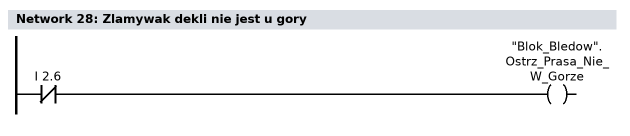
NETWORK
TITLE = Zlamywak dekli nie jest u gory 
      AN    I 2.6;
      =     "Blok_Bledow".Ostrz_Prasa_Nie_W_Gorze;
END_FUNCTION

FUNCTION "FC_HMI" : VOID	// FC 120
VERSION : 0.1
VAR_TEMP
  LW0_Help : INT ;
END_VAR
BEGIN
NETWORK
TITLE =
//Ten network celowo wolny
NETWORK
TITLE = Tryb Pracy Wiazanie poprzeczne
//Wybranie trybu pracy resetuje pozostale tryby pracy
//1-Przelot
      A     "DB_HMI".HMI_IN_OUT.Tp_Przelot;
      R     "DB_HMI".HMI_IN_OUT.Tp_Wiazanie_Poprzeczne;
      R     "DB_HMI".HMI_IN_OUT.Tp_Wiazanie_Wzdluzne;
      R     "DB_HMI".HMI_IN_OUT.Tp_Wiazanie_Pop_Wzdl;
      R     "Blok_Para".Wiazanie_Poprzeczne;
      R     "Blok_Para".Wiazanie_Wzdluzne;
NETWORK
TITLE = Tryb Pracy Wiazanie poprzeczne
//Wybranie trybu pracy resetuje pozostale tryby pracy
//2-Wiazanie Poprzeczne
      A     "DB_HMI".HMI_IN_OUT.Tp_Wiazanie_Poprzeczne;
      R     "DB_HMI".HMI_IN_OUT.Tp_Przelot;
      R     "DB_HMI".HMI_IN_OUT.Tp_Wiazanie_Wzdluzne;
      R     "DB_HMI".HMI_IN_OUT.Tp_Wiazanie_Pop_Wzdl;
      S     "Blok_Para".Wiazanie_Poprzeczne;
      R     "Blok_Para".Wiazanie_Wzdluzne;
NETWORK
TITLE = Tryb Pracy Wiazanie poprzeczne
//Wybranie trybu pracy resetuje pozostale tryby pracy
//3-Wiazanie Wzdluzne
      A     "DB_HMI".HMI_IN_OUT.Tp_Wiazanie_Wzdluzne;
      R     "DB_HMI".HMI_IN_OUT.Tp_Przelot;
      R     "DB_HMI".HMI_IN_OUT.Tp_Wiazanie_Poprzeczne;
      R     "DB_HMI".HMI_IN_OUT.Tp_Wiazanie_Pop_Wzdl;
      R     "Blok_Para".Wiazanie_Poprzeczne;
      S     "Blok_Para".Wiazanie_Wzdluzne;
NETWORK
TITLE = Tryb Pracy Wiazanie poprzeczne
//Wybranie trybu pracy resetuje pozostale tryby pracy
//4-Wiazanie Poprzeczne i wzdluzne
      A     "DB_HMI".HMI_IN_OUT.Tp_Wiazanie_Pop_Wzdl;
      R     "DB_HMI".HMI_IN_OUT.Tp_Przelot;
      R     "DB_HMI".HMI_IN_OUT.Tp_Wiazanie_Poprzeczne;
      R     "DB_HMI".HMI_IN_OUT.Tp_Wiazanie_Wzdluzne;
      S     "Blok_Para".Wiazanie_Poprzeczne;
      S     "Blok_Para".Wiazanie_Wzdluzne;
NETWORK
TITLE = wybrano tryb pracy przelot
      AN    "Blok_Para".Wiazanie_Wzdluzne;
      AN    "Blok_Para".Wiazanie_Poprzeczne;
      =     "DB_HMI".HMI_IN.Wybrano_TP_Przelot;
//-wzdl
      A     "Blok_Para".Wiazanie_Wzdluzne;
      AN    "Blok_Para".Wiazanie_Poprzeczne;
      =     "DB_HMI".HMI_IN.Wybrano_TP_Wiazanie_Wzdl;
//-pop
      AN    "Blok_Para".Wiazanie_Wzdluzne;
      A     "Blok_Para".Wiazanie_Poprzeczne;
      =     "DB_HMI".HMI_IN.Wybrano_TP_Wiazanie_Pop;
//-pop -wzdl
      A     "Blok_Para".Wiazanie_Wzdluzne;
      A     "Blok_Para".Wiazanie_Poprzeczne;
      =     "DB_HMI".HMI_IN.Wybrano_TP_Wiazanie_Krzy;
NETWORK
TITLE =
//znacznik trybu wiazania
//krok_1  - przelot
      A     "DB_HMI".HMI_IN.Wybrano_TP_Przelot;
      L     1;
      JC    ztw;
//krok_2 - wzdluzna
      A     "DB_HMI".HMI_IN.Wybrano_TP_Wiazanie_Wzdl;
      L     2;
      JC    ztw;
//krok_3 - poprzeczne
      A     "DB_HMI".HMI_IN.Wybrano_TP_Wiazanie_Pop;
      L     3;
      JC    ztw;
//krok_4 - krzyzowe
      A     "DB_HMI".HMI_IN.Wybrano_TP_Wiazanie_Krzy;
      L     4;
      JC    ztw;
//daj 0
ztw:  T     "DB_HMI".HMI_IN.tryb_wiaz;
NETWORK
TITLE = Tryb Pracy Wiazanie wzduzne
//Zalaczenie Pozycjonowania
      A     "DB_HMI".HMI_IN_OUT.Tp_Pozycjonowanie;
      S     "Blok_Para".Pozycjonowanie;
      AN    "DB_HMI".HMI_IN_OUT.Tp_Pozycjonowanie;
      R     "Blok_Para".Pozycjonowanie;
      NOP   0;
NETWORK
TITLE = fotokomorka hamowania obrotnicy do kata 0st
//Fotokomorki katow pozycjonowania obrotnicy
      A     "AIO".Czuj_19_B.Czujnik_Ham_0_St;
      =     "DB_HMI".HMI_IN.Czujnik_Ham_0_St;
      A     "AIO".Czuj_19_B.Czujnik_0_St;
      =     "DB_HMI".HMI_IN.Czujnik_0_St;
      A     "AIO".Czuj_19_B.Czujnik_Ham_90_St;
      =     "DB_HMI".HMI_IN.Czujnik_Ham_90_St;
      A     "AIO".Czuj_19_B.Czujnik_90_St;
      =     "DB_HMI".HMI_IN.Czujnik_90_St;
      A     "AIO".Czuj_17_B.Czujnik_Ham_180_St;
      =     "DB_HMI".HMI_IN.Czujnik_Ham_180_St;
      A     "AIO".Czuj_17_B.Czujnik_180_St;
      =     "DB_HMI".HMI_IN.Czujnik_180_St;
      A     "AIO".Czuj_17_B.Czujnik_Ham_270_St;
      =     "DB_HMI".HMI_IN.Czujnik_Ham_270_St;
      A     "AIO".Czuj_17_B.Czujnik_270_St;
      =     "DB_HMI".HMI_IN.Czujnik_270_St;
NETWORK
TITLE = foto przednie bandzie wlotowej
//Fotokommorki
      A     "AIO".Banda_23.Foto_1;
      =     "DB_HMI".HMI_IN.Foto_Tasma_1_Przod;
      A     "AIO".Banda_23.Foto_2;
      =     "DB_HMI".HMI_IN.Foto_Tasma_1_Tyl;
      A     "AIO".Banda_24.Foto_1;
      =     "DB_HMI".HMI_IN.Foto_Tasma_2_Przod;
      A     "AIO".Banda_24.Foto_2;
      =     "DB_HMI".HMI_IN.Foto_Tasma_2_Tyl;
      A     "AIO".Obr_15.Foto_1;
      =     "DB_HMI".HMI_IN.Foto_Obrotnica_3_Przod;
      A     "AIO".Obr_15.Foto_2;
      =     "DB_HMI".HMI_IN.Foto_Obrotnica_3_Tyl;
      A     "AIO".Banda_2.Foto_1;
      =     "DB_HMI".HMI_IN.Foto_Tasma_4_Przod;
      A     "AIO".Banda_2.Foto_2;
      =     "DB_HMI".HMI_IN.Foto_Tasma_4_Tyl;
NETWORK
TITLE = tasma 1
//do wizualizacji przemieszczania palety na tasmie 1
      AN    "AIO".Banda_23.Foto_1;
      A     "AIO".Banda_23.Foto_2;
      =     "DB_HMI".HMI_IN.Paleta_na_Tasmie_1_T;
      A     "AIO".Banda_23.Foto_1;
      AN    "AIO".Banda_23.Foto_2;
      AN    "AIO".Banda_24.Foto_2;
      =     "DB_HMI".HMI_IN.Paleta_na_Tasmie_1_P;
      A     "AIO".Banda_23.Foto_1;
      A     "AIO".Banda_23.Foto_2;
      =     "DB_HMI".HMI_IN.Paleta_na_Tasmie_1;
NETWORK
TITLE = tasma 2
//do wizualizacji przemieszczania palety na tasmie 2
      AN    "AIO".Banda_24.Foto_1;
      A     "AIO".Banda_24.Foto_2;
      =     "DB_HMI".HMI_IN.Paleta_na_Tasmie_2_T;
      A     "AIO".Banda_24.Foto_1;
      AN    "AIO".Banda_24.Foto_2;
      AN    "AIO".Obr_15.Foto_1;
      =     "DB_HMI".HMI_IN.Paleta_na_Tasmie_2_P;
      A     "AIO".Banda_24.Foto_1;
      A     "AIO".Banda_24.Foto_2;
      =     "DB_HMI".HMI_IN.Paleta_na_Tasmie_2;
NETWORK
TITLE = tasma 3 (obrotnica)
//do wizualizacji przemieszczania palety na tasmie 3
      A     "AIO".Obr_15.Foto_1;
      AN    "AIO".Obr_15.Foto_2;
      A     "DB_HMI".HMI_IN.Czujnik_0_St;
      =     "DB_HMI".HMI_IN.Paleta_na_Tasmie_3_T;
      AN    "AIO".Obr_15.Foto_1;
      A     "AIO".Obr_15.Foto_2;
      AN    "AIO".Banda_2.Foto_2;
      A     "DB_HMI".HMI_IN.Czujnik_0_St;
      =     "DB_HMI".HMI_IN.Paleta_na_Tasmie_3_P;
      A     "AIO".Obr_15.Foto_1;
      A     "AIO".Obr_15.Foto_2;
      A(;
      O     "DB_HMI".HMI_IN.Czujnik_0_St;
      O     "DB_HMI".HMI_IN.Czujnik_180_St;
      );
      =     "DB_HMI".HMI_IN.Paleta_na_Tasmie_3_0_180;
      A     "AIO".Obr_15.Foto_1;
      A     "AIO".Obr_15.Foto_2;
      A(;
      O     "DB_HMI".HMI_IN.Czujnik_90_St;
      O     "DB_HMI".HMI_IN.Czujnik_270_St;
      );
      =     "DB_HMI".HMI_IN.Paleta_na_Tasmie_3_90_27;
NETWORK
TITLE = tasma 4
//do wizualizacji przemieszczania palety na tasmie 4
      AN    "AIO".Banda_2.Foto_1;
      A     "AIO".Banda_2.Foto_2;
      =     "DB_HMI".HMI_IN.Paleta_na_Tasmie_4_T;
      A     "AIO".Banda_2.Foto_1;
      AN    "AIO".Banda_2.Foto_2;
      =     "DB_HMI".HMI_IN.Paleta_na_Tasmie_4_P;
      A     "AIO".Banda_2.Foto_1;
      A     "AIO".Banda_2.Foto_2;
      =     "DB_HMI".HMI_IN.Paleta_na_Tasmie_4;
NETWORK
TITLE = motor obrotnica 3 counter clock wise
//Napedy band
      A     "AIO".Obr_15.CC_Wise;
      =     "DB_HMI".HMI_IN.Motor_Obrotnica_3_CCW;
      A     "AIO".Obr_15.C_Wise;
      =     "DB_HMI".HMI_IN.Motor_Obrotnica_3_CW;
      A     "AIO".Banda_23.CC_Wise;
      =     "DB_HMI".HMI_IN.Motor_Tasma_1_Przod;
      A     "AIO".Banda_23.C_Wise;
      =     "DB_HMI".HMI_IN.Motor_Tasma_1_Tyl;
      A     "AIO".Banda_24.C_Wise;
      =     "DB_HMI".HMI_IN.Motor_Tasma_2_Przod;
      A     "AIO".Banda_24.CC_Wise;
      =     "DB_HMI".HMI_IN.Motor_Tasma_2_Tyl;
      A     "AIO".Banda_1.C_Wise;
      =     "DB_HMI".HMI_IN.Motor_Tasma_3_Przod;
      A     "AIO".Banda_1.CC_Wise;
      =     "DB_HMI".HMI_IN.Motor_Tasma_3_Tyl;
      A     "AIO".Banda_2.CC_Wise;
      =     "DB_HMI".HMI_IN.Motor_Tasma_4_Przod;
      A     "AIO".Banda_2.C_Wise;
      =     "DB_HMI".HMI_IN.Motor_Tasma_4_Tyl;
NETWORK
TITLE = obwod bezpieczenstwa bindownicy
//sygnaly wymiany danych pomiedzy transportem palet a bindownica
      A     I 2.0;
      =     "DB_HMI".HMI_IN.Interfefs_B_do_TP_B1;
      A     I 2.1;
      =     "DB_HMI".HMI_IN.Interfefs_B_do_TP_B2;
      A     I 2.3;
      =     "DB_HMI".HMI_IN.Interfefs_B_do_TP_B3;
      A     I 2.4;
      =     "DB_HMI".HMI_IN.Interfefs_B_do_TP_B4;
      A     I 2.2;
      =     "DB_HMI".HMI_IN.Interfefs_B_do_TP_B5;
//Transport do bindownicy 
      A     M 6.3;
      =     "DB_HMI".HMI_IN.Interfefs_TP_do_B_TP1;
      A     Q 1.1;
      =     "DB_HMI".HMI_IN.Interfefs_TP_do_B_TP2;
      A     Q 1.2;
      =     "DB_HMI".HMI_IN.Interfefs_TP_do_B_TP3;
NETWORK
TITLE = przycisk zalaczenie Strefy bezpieczenstwa
//przyciski, przelaczniki kierunkow i lampki na panelu
      A     I 0.0;
      =     "DB_HMI".HMI_IN.PB_Strefa_bezpieczenstwa;
      A     I 0.1;
      =     "DB_HMI".HMI_IN.PB_Reczny;
      A     I 0.2;
      =     "DB_HMI".HMI_IN.PB_Auto;
      A     I 0.3;
      =     "DB_HMI".HMI_IN.PB_Reset;
      A     I 0.4;
      =     "DB_HMI".HMI_IN.PB_Stop;
      A     I 0.5;
      =     "DB_HMI".HMI_IN.PB_Cykl_Start;
      A     I 0.6;
      =     "DB_HMI".HMI_IN.PB_Tasma1_Tyl;
      A     I 0.7;
      =     "DB_HMI".HMI_IN.PB_Tasma1_Przod;
      A     I 1.0;
      =     "DB_HMI".HMI_IN.PB_Tasma2_Tyl;
      A     I 1.1;
      =     "DB_HMI".HMI_IN.PB_Tasma2_Przod;
      A     I 1.2;
      =     "DB_HMI".HMI_IN.PB_Tasma3_Tyl;
      A     I 1.3;
      =     "DB_HMI".HMI_IN.PB_Tasma3_Przod;
      A     I 1.4;
      =     "DB_HMI".HMI_IN.PB_Tasma4_Tyl;
      A     I 1.5;
      =     "DB_HMI".HMI_IN.PB_Tasma4_Przod;
      A     I 1.6;
      =     "DB_HMI".HMI_IN.PB_Tasma3_Obr_CW;
      A     I 1.7;
      =     "DB_HMI".HMI_IN.PB_Tasma3_Obr_CCW;
      A     Q 0.0;
      =     "DB_HMI".HMI_IN.Lampka_Blad_Bind;
      A     Q 0.1;
      =     "DB_HMI".HMI_IN.Lampka_Strzal_Tasmy;
      A     Q 0.2;
      =     "DB_HMI".HMI_IN.Lampka_Strefa_Bezp;
      A     Q 0.3;
      =     "DB_HMI".HMI_IN.Lampka_PB_Reczny;
      A     Q 0.4;
      =     "DB_HMI".HMI_IN.Lampka_PB_Auto;
      A     Q 0.5;
      =     "DB_HMI".HMI_IN.Lampka_PB_Reset;
      A     Q 0.6;
      =     "DB_HMI".HMI_IN.Lampka_PB_Stop;
      A     Q 0.7;
      =     "DB_HMI".HMI_IN.Lampka_PB_Cykl_Start;
NETWORK
TITLE =
//Start/Stop calej lini
      A     "DB_HMI".HMI_OUT.Start_Lini_z_OP;
      =     "Blok_Para".Start_Lini_z_OP;
      A     "DB_HMI".HMI_OUT.Stop_Lini_z_OP;
      =     "Blok_Para".Stop_Lini_z_OP;
NETWORK
TITLE = //wyjazd wtrybie auto
//Wyzwolenie wyjazdu palety gdy paleta stoi na bandzie obrotowej a nie wyjezdza
//
      A     "DB_HMI".HMI_OUT.Wyzwolenie_Wyjazdu;
      =     "Blok_Para".Trigger_Wyjazd;
NETWORK
TITLE = Znacznik stanu kurtyny optycznej na wlocie
//Bariery optyczne bindownicy
      AN    "AIO".Kurtyna_25.OSSD_Tor_1_1;
      AN    "AIO".Kurtyna_25.OSSD_Tor_1_2;
      AN    "AIO".Kurtyna_25.OSSD_Tor_2_1;
      AN    "AIO".Kurtyna_25.OSSD_Tor_2_2;
      =     "DB_HMI".HMI_IN.Kurtyna_Wlot_Ok;
      AN    "AIO".Kurtyna_26.OSSD_Tor_1_1;
      AN    "AIO".Kurtyna_26.OSSD_Tor_1_2;
      AN    "AIO".Kurtyna_26.OSSD_Tor_2_1;
      AN    "AIO".Kurtyna_26.OSSD_Tor_2_2;
      =     "DB_HMI".HMI_IN.Kurtyna_Wylot_Ok;
      A     M 6.2;
      =     "DB_HMI".HMI_IN.Rygiel;
NETWORK
TITLE = Znacznik pracy calej linii transportowej
      A     Q 8.3;
      =     "DB_HMI".HMI_IN.Linia_transportowa_praca;
NETWORK
TITLE = tryb pracy bindownicy: Auto(1) Reczny(0)
      A     "Blok_Bledow_Program".Blad_Krok_1;
      =     "DB_HMI".HMI_IN.Krok_1;
      A     "Blok_Bledow_Program".Blad_Krok_2;
      =     "DB_HMI".HMI_IN.Krok_2;
      A     "Blok_Bledow_Program".Blad_Krok_3;
      =     "DB_HMI".HMI_IN.Krok_3;
      A     "Blok_Bledow_Program".Blad_Krok_4;
      =     "DB_HMI".HMI_IN.Krok_4;
      A     "Blok_Bledow_Program".Blad_Krok_5;
      =     "DB_HMI".HMI_IN.Krok_5;
      A     "Blok_Bledow_Program".Blad_Krok_6;
      =     "DB_HMI".HMI_IN.Krok_6;
NETWORK
TITLE =
//przypisanie stanu wejsc i wyjsc
      L     IB 0;
      T     "DB_HMI".HMI_IN.input_0;
      L     IB 1;
      T     "DB_HMI".HMI_IN.input_1;
      L     IB 2;
      T     "DB_HMI".HMI_IN.input_2;
      L     IB 3;
      T     "DB_HMI".HMI_IN.input_3;
      L     QB 0;
      T     "DB_HMI".HMI_IN.output_0;
      L     QB 1;
      T     "DB_HMI".HMI_IN.output_1;
      L     QB 2;
      T     "DB_HMI".HMI_IN.output_2;
      L     QB 3;
      T     "DB_HMI".HMI_IN.output_3;
      L     IB 8;
      T     "DB_HMI".HMI_IN.input_8;
      L     IB 9;
      T     "DB_HMI".HMI_IN.input_9;
      L     IB 10;
      T     "DB_HMI".HMI_IN.input_10;
      L     IB 11;
      T     "DB_HMI".HMI_IN.input_11;
NETWORK
TITLE = krok 1 trybu pracy
//Przypisanie aktualnych krokow 
//krok_1  - jedz na pozycje 
      A     "Blok_Para".Krok_1;
      L     1;
      JC    tr;
//krok_2 - szukaj srodka 
      A     "Blok_Para".krok_2;
      L     2;
      JC    tr;
//krok_3 - jedz na prawo
      A     "Blok_Para".krok_3;
      L     3;
      JC    tr;
//krok_4 - strzelaj 
      A     "Blok_Para".krok_4;
      L     4;
      JC    tr;
//krok_5  - pauza po strzale
      A     "Blok_Para".krok_5;
      L     5;
      JC    tr;
//krok_6 - jedz do srodka
      A     "Blok_Para".krok_6;
      L     6;
      JC    tr;
//daj 0
      L     0;
tr:   T     "DB_HMI".HMI_IN.INT_Liczba_Akt_Kroku;
NETWORK
TITLE = znacznik migania bledu
//Sprawdzenie czy sa bledy jak sa to miganie bledow
      SET;
      R     "DB_HMI".HMI_IN.Znacznik_Migania_Bledu;
      O(;
      L     DB119.DBD 0;
      L     0;
      <>D;
      );
      O(;
      L     DB119.DBD 4;
      L     0;
      <>D;
      );
      O(;
      L     DB119.DBD 8;
      L     0;
      <>D;
      );
      S     "DB_HMI".HMI_IN.Znacznik_Migania_Bledu;
NETWORK
TITLE = czujnik prasy s 22
//Obsluga wygladu prasy
//
      A     I 2.6;
      =     "DB_HMI".HMI_IN.Czujnik_Prasa;
//zawor prasa
      AN    Q 1.0;
      =     "DB_HMI".HMI_IN.Stan_Zaworu;
NETWORK
TITLE =
//Aktualizacja godziny/daty panela z godzina/czasem PLC
      CALL  "READ_CLK" (
           RET_VAL                  := #LW0_Help,
           CDT                      := "DB_HMI".HMI_IN.Aktualna_Data);
END_FUNCTION

FUNCTION "Funkcja_Zegara" : VOID	// FC 140
AUTHOR : Kng
NAME : HELP_FC
VERSION : 0.1
VAR_INPUT
  Timer_NR : TIMER ;
  Czas : S5TIME ;
END_VAR
VAR_IN_OUT
  Wyjscie : BOOL ;
END_VAR
BEGIN
NETWORK
TITLE =
      A     #Timer_NR;
      SAVE;
      NOT;
      L     #Czas;
      SD    #Timer_NR;
      X     BR;
      X     #Wyjscie;
      =     #Wyjscie;
END_FUNCTION

DATA_BLOCK DB 4
VERSION : 0.0
"Czesc_Bindujaca"
BEGIN
END_DATA_BLOCK

DATA_BLOCK DB 5
VERSION : 0.0
"Czesc_Trasnportujaca"
BEGIN
END_DATA_BLOCK

DATA_BLOCK "AIO"	// DB 10
VERSION : 0.1
  STRUCT
   Banda_1 : UDT 1;	//Temporary placeholder variable
   Banda_2 : UDT 1;
   Banda_3 : UDT 1;
   Banda_4 : UDT 9;
   Banda_5 : UDT 1;
   Banda_6 : UDT 1;
   Banda_7 : UDT 1;
   Banda_8 : UDT 1;
   Banda_9 : UDT 1;
   Banda_10 : UDT 1;
   Banda_11 : UDT 1;
   Banda_12 : UDT 1;
   Banda_13 : UDT 9;
   Banda_14 : UDT 1;
   Obr_15 : UDT 11;
   Czuj_19_B : UDT 7;
   Czuj_17_B : UDT 10;
   Obr_18 : UDT 6;
   Czuj_19 : UDT 7;
   Obr_20 : UDT 6;
   Czuj_21 : UDT 7;
   Czuj_22 : UDT 8;
   Banda_23 : UDT 1;
   Banda_24 : UDT 1;
   Kurtyna_25 : UDT 2;
   Kurtyna_26 : UDT 2;
   ESTOP_27 : UDT 3;
   ESTOP_28 : UDT 3;
   ESTOP_29 : UDT 3;
   ESTOP_30 : UDT 3;
   ESTOP_31 : UDT 3;
   Rygiel_16 : UDT 2;
   Reset_17 : UDT 12;
  END_STRUCT ;	
BEGIN
END_DATA_BLOCK

DATA_BLOCK "Blok_Para"	// DB 12
VERSION : 0.1
  STRUCT
   Wiazanie_Poprzeczne : BOOL ;	//Wiaz wzdluz
   Wiazanie_Wzdluzne : BOOL ;
   Pozycjonowanie : BOOL ;
   Przelacz_Na_Auto : BOOL ;	//warunkowe przejscie na auto
   Start_Lini_z_OP : BOOL ;
   Stop_Lini_z_OP : BOOL ;
   Trigger_Wyjazd : BOOL ;	////wyjazd wtrybie auto
   Ser_Pokrycie_Foto : BOOL ;
   Pozycjon_Banda_Lewo : BOOL ;
   Pozycjon_Banda_Prawo : BOOL ;
   Pozycjon_Banda_Srodek : BOOL ;	//rozakaz pozycjonowana
   Banda_Poz_Lewa : BOOL ;
   Banda_Poz_Prawa : BOOL ;
   Banda_Poz_Srodek : BOOL ;
   Banda_Poz_Potw : BOOL ;
   Jedz_Na_0st : BOOL ;
   Jedz_Na_90st : BOOL ;
   Jedz_Na_180st : BOOL ;
   Jedz_Na_270st : BOOL ;
   Poz_0_st : BOOL ;
   Poz_90_st : BOOL ;
   Poz_180_st : BOOL ;
   Poz_270_st : BOOL ;
   Poz_Obr_Osiagnieta : BOOL ;
   Odblokuj_Rolki : BOOL ;
   Odblokuj_Obrotnice : BOOL ;
   Poz_Obr_Osiagnieta1 : BOOL ;
   Pozycja_Obrotnicy : INT ;
   Bin_Licznik : INT ;	//licznik bindownicy
   Rezerwa_Para : DWORD ;
   Krok_1 : BOOL ;
   krok_2 : BOOL ;
   krok_3 : BOOL ;
   krok_4 : BOOL ;
   krok_5 : BOOL ;
   krok_6 : BOOL ;
   krok_7 : BOOL ;
   krok_8 : BOOL ;
   krok_9 : BOOL ;
  END_STRUCT ;	
BEGIN
END_DATA_BLOCK

DATA_BLOCK "Blok_Bledow_Program"	// DB 13
VERSION : 0.1
  STRUCT
   Blad_Krok_1 : BOOL ;	//Blad kroku nr 1 (Przekrokczony czas jazdy  na zadana pozycje)
   Blad_Krok_2 : BOOL ;	//Blad kroku nr 2 (Przekrokczony czas szukania srodka palety)
   Blad_Krok_3 : BOOL ;	//Blad kroku nr 3 (Przekrokczony czas pozycjonowania palety lewo/prawo)
   Blad_Krok_4 : BOOL ;	//Blad kroku nr 4 (Przekrokczony czas strzalu bindownicy)
   Blad_Krok_5 : BOOL ;	//Blad kroku nr 6 (Przekrokczony czas czasu postoju)
   Blad_Krok_6 : BOOL ;	//Blad kroku nr 5 (Przekrokczony czas powrotu lewo/prawo)
   Blad_Krok_7 : BOOL ;	//Rezerwa
   Blad_Krok_8 : BOOL ;	//Rezerwa
   Blad_Krok_9 : BOOL ;	//Rezerwa
   Blad_Krok_10 : BOOL ;	//Rezerwa
  END_STRUCT ;	
BEGIN
END_DATA_BLOCK

DATA_BLOCK "Asi_input"	// DB 80
VERSION : 0.1
  STRUCT
   Adres_1_bit_0 : BOOL ;	//Temporary placeholder variable
   Adres_1_bit_1 : BOOL ;
   Adres_1_bit_2 : BOOL ;
   Adres_1_bit_3 : BOOL ;
   Adres_0_bit_0 : BOOL ;	//Temporary placeholder variable
   Adres_0_bit_1 : BOOL ;
   Adres_0_bit_2 : BOOL ;
   Adres_0_bit_3 : BOOL ;
   Adres_3_bit_0 : BOOL ;	//Temporary placeholder variable
   Adres_3_bit_1 : BOOL ;
   Adres_3_bit_2 : BOOL ;
   Adres_3_bit_3 : BOOL ;
   Adres_2_bit_0 : BOOL ;	//Temporary placeholder variable
   Adres_2_bit_1 : BOOL ;
   Adres_2_bit_2 : BOOL ;
   Adres_2_bit_3 : BOOL ;
   Adres_5_bit_0 : BOOL ;	//Temporary placeholder variable
   Adres_5_bit_1 : BOOL ;
   Adres_5_bit_2 : BOOL ;
   Adres_5_bit_3 : BOOL ;
   Adres_4_bit_0 : BOOL ;	//Temporary placeholder variable
   Adres_4_bit_1 : BOOL ;
   Adres_4_bit_2 : BOOL ;
   Adres_4_bit_3 : BOOL ;
   Adres_7_bit_0 : BOOL ;	//Temporary placeholder variable
   Adres_7_bit_1 : BOOL ;
   Adres_7_bit_2 : BOOL ;
   Adres_7_bit_3 : BOOL ;
   Adres_6_bit_0 : BOOL ;	//Temporary placeholder variable
   Adres_6_bit_1 : BOOL ;
   Adres_6_bit_2 : BOOL ;
   Adres_6_bit_3 : BOOL ;
   Adres_9_bit_0 : BOOL ;	//Temporary placeholder variable
   Adres_9_bit_1 : BOOL ;
   Adres_9_bit_2 : BOOL ;
   Adres_9_bit_3 : BOOL ;
   Adres_8_bit_0 : BOOL ;	//Temporary placeholder variable
   Adres_8_bit_1 : BOOL ;
   Adres_8_bit_2 : BOOL ;
   Adres_8_bit_3 : BOOL ;
   Adres_11_bit_0 : BOOL ;	//Temporary placeholder variable
   Adres_11_bit_1 : BOOL ;
   Adres_11_bit_2 : BOOL ;
   Adres_11_bit_3 : BOOL ;
   Adres_10_bit_0 : BOOL ;	//Temporary placeholder variable
   Adres_10_bit_1 : BOOL ;
   Adres_10_bit_2 : BOOL ;
   Adres_10_bit_3 : BOOL ;
   Adres_13_bit_0 : BOOL ;	//Temporary placeholder variable
   Adres_13_bit_1 : BOOL ;
   Adres_13_bit_2 : BOOL ;
   Adres_13_bit_3 : BOOL ;
   Adres_12_bit_0 : BOOL ;	//Temporary placeholder variable
   Adres_12_bit_1 : BOOL ;
   Adres_12_bit_2 : BOOL ;
   Adres_12_bit_3 : BOOL ;
   Adres_15_bit_0 : BOOL ;	//Temporary placeholder variable
   Adres_15_bit_1 : BOOL ;
   Adres_15_bit_2 : BOOL ;
   Adres_15_bit_3 : BOOL ;
   Adres_14_bit_0 : BOOL ;	//Temporary placeholder variable
   Adres_14_bit_1 : BOOL ;
   Adres_14_bit_2 : BOOL ;
   Adres_14_bit_3 : BOOL ;
   Adres_17_bit_0 : BOOL ;	//Temporary placeholder variable
   Adres_17_bit_1 : BOOL ;
   Adres_17_bit_2 : BOOL ;
   Adres_17_bit_3 : BOOL ;
   Adres_16_bit_0 : BOOL ;	//Temporary placeholder variable
   Adres_16_bit_1 : BOOL ;
   Adres_16_bit_2 : BOOL ;
   Adres_16_bit_3 : BOOL ;
   Adres_19_bit_0 : BOOL ;	//Temporary placeholder variable
   Adres_19_bit_1 : BOOL ;
   Adres_19_bit_2 : BOOL ;
   Adres_19_bit_3 : BOOL ;
   Adres_18_bit_0 : BOOL ;	//Temporary placeholder variable
   Adres_18_bit_1 : BOOL ;
   Adres_18_bit_2 : BOOL ;
   Adres_18_bit_3 : BOOL ;
   Adres_21_bit_0 : BOOL ;	//Temporary placeholder variable
   Adres_21_bit_1 : BOOL ;
   Adres_21_bit_2 : BOOL ;
   Adres_21_bit_3 : BOOL ;
   Adres_20_bit_0 : BOOL ;	//Temporary placeholder variable
   Adres_20_bit_1 : BOOL ;
   Adres_20_bit_2 : BOOL ;
   Adres_20_bit_3 : BOOL ;
   Adres_23_bit_0 : BOOL ;	//Temporary placeholder variable
   Adres_23_bit_1 : BOOL ;
   Adres_23_bit_2 : BOOL ;
   Adres_23_bit_3 : BOOL ;
   Adres_22_bit_0 : BOOL ;	//Temporary placeholder variable
   Adres_22_bit_1 : BOOL ;
   Adres_22_bit_2 : BOOL ;
   Adres_22_bit_3 : BOOL ;
   Adres_25_bit_0 : BOOL ;	//Temporary placeholder variable
   Adres_25_bit_1 : BOOL ;
   Adres_25_bit_2 : BOOL ;
   Adres_25_bit_3 : BOOL ;
   Adres_24_bit_0 : BOOL ;	//Temporary placeholder variable
   Adres_24_bit_1 : BOOL ;
   Adres_24_bit_2 : BOOL ;
   Adres_24_bit_3 : BOOL ;
   Adres_27_bit_0 : BOOL ;	//Temporary placeholder variable
   Adres_27_bit_1 : BOOL ;
   Adres_27_bit_2 : BOOL ;
   Adres_27_bit_3 : BOOL ;
   Adres_26_bit_0 : BOOL ;	//Temporary placeholder variable
   Adres_26_bit_1 : BOOL ;
   Adres_26_bit_2 : BOOL ;
   Adres_26_bit_3 : BOOL ;
   Adres_29_bit_0 : BOOL ;	//Temporary placeholder variable
   Adres_29_bit_1 : BOOL ;
   Adres_29_bit_2 : BOOL ;
   Adres_29_bit_3 : BOOL ;
   Adres_28_bit_0 : BOOL ;	//Temporary placeholder variable
   Adres_28_bit_1 : BOOL ;
   Adres_28_bit_2 : BOOL ;
   Adres_28_bit_3 : BOOL ;
   Adres_31_bit_0 : BOOL ;	//Temporary placeholder variable
   Adres_31_bit_1 : BOOL ;
   Adres_31_bit_2 : BOOL ;
   Adres_31_bit_3 : BOOL ;
   Adres_30_bit_0 : BOOL ;	//Temporary placeholder variable
   Adres_30_bit_1 : BOOL ;
   Adres_30_bit_2 : BOOL ;
   Adres_30_bit_3 : BOOL ;
   B_Adres_1_bit_0 : BOOL ;	//Temporary placeholder variable
   B_Adres_1_bit_1 : BOOL ;
   B_Adres_1_bit_2 : BOOL ;
   B_Adres_1_bit_3 : BOOL ;
   B_Adres_0_bit_0 : BOOL ;
   B_Adres_0_bit_1 : BOOL ;
   B_Adres_0_bit_2 : BOOL ;
   B_Adres_0_bit_3 : BOOL ;
   B_Adres_3_bit_0 : BOOL ;	//Temporary placeholder variable
   B_Adres_3_bit_1 : BOOL ;
   B_Adres_3_bit_2 : BOOL ;
   B_Adres_3_bit_3 : BOOL ;
   B_Adres_2_bit_0 : BOOL ;	//Temporary placeholder variable
   B_Adres_2_bit_1 : BOOL ;
   B_Adres_2_bit_2 : BOOL ;
   B_Adres_2_bit_3 : BOOL ;
   B_Adres_5_bit_0 : BOOL ;	//Temporary placeholder variable
   B_Adres_5_bit_1 : BOOL ;
   B_Adres_5_bit_2 : BOOL ;
   B_Adres_5_bit_3 : BOOL ;
   B_Adres_4_bit_0 : BOOL ;	//Temporary placeholder variable
   B_Adres_4_bit_1 : BOOL ;
   B_Adres_4_bit_2 : BOOL ;
   B_Adres_4_bit_3 : BOOL ;
   B_Adres_7_bit_0 : BOOL ;	//Temporary placeholder variable
   B_Adres_7_bit_1 : BOOL ;
   B_Adres_7_bit_2 : BOOL ;
   B_Adres_7_bit_3 : BOOL ;
   B_Adres_6_bit_0 : BOOL ;	//Temporary placeholder variable
   B_Adres_6_bit_1 : BOOL ;
   B_Adres_6_bit_2 : BOOL ;
   B_Adres_6_bit_3 : BOOL ;
   B_Adres_9_bit_0 : BOOL ;	//Temporary placeholder variable
   B_Adres_9_bit_1 : BOOL ;
   B_Adres_9_bit_2 : BOOL ;
   B_Adres_9_bit_3 : BOOL ;
   B_Adres_8_bit_0 : BOOL ;	//Temporary placeholder variable
   B_Adres_8_bit_1 : BOOL ;
   B_Adres_8_bit_2 : BOOL ;
   B_Adres_8_bit_3 : BOOL ;
   B_Adres_11_bit_0 : BOOL ;	//Temporary placeholder variable
   B_Adres_11_bit_1 : BOOL ;
   B_Adres_11_bit_2 : BOOL ;
   B_Adres_11_bit_3 : BOOL ;
   B_Adres_10_bit_0 : BOOL ;	//Temporary placeholder variable
   B_Adres_10_bit_1 : BOOL ;
   B_Adres_10_bit_2 : BOOL ;
   B_Adres_10_bit_3 : BOOL ;
   B_Adres_13_bit_0 : BOOL ;	//Temporary placeholder variable
   B_Adres_13_bit_1 : BOOL ;
   B_Adres_13_bit_2 : BOOL ;
   B_Adres_13_bit_3 : BOOL ;
   B_Adres_12_bit_0 : BOOL ;	//Temporary placeholder variable
   B_Adres_12_bit_1 : BOOL ;
   B_Adres_12_bit_2 : BOOL ;
   B_Adres_12_bit_3 : BOOL ;
   B_Adres_15_bit_0 : BOOL ;	//Temporary placeholder variable
   B_Adres_15_bit_1 : BOOL ;
   B_Adres_15_bit_2 : BOOL ;
   B_Adres_15_bit_3 : BOOL ;
   B_Adres_14_bit_0 : BOOL ;	//Temporary placeholder variable
   B_Adres_14_bit_1 : BOOL ;
   B_Adres_14_bit_2 : BOOL ;
   B_Adres_14_bit_3 : BOOL ;
   B_Adres_17_bit_0 : BOOL ;	//Temporary placeholder variable
   B_Adres_17_bit_1 : BOOL ;
   B_Adres_17_bit_2 : BOOL ;
   B_Adres_17_bit_3 : BOOL ;
   B_Adres_16_bit_0 : BOOL ;	//Temporary placeholder variable
   B_Adres_16_bit_1 : BOOL ;
   B_Adres_16_bit_2 : BOOL ;
   B_Adres_16_bit_3 : BOOL ;
   B_Adres_19_bit_0 : BOOL ;	//Temporary placeholder variable
   B_Adres_19_bit_1 : BOOL ;
   B_Adres_19_bit_2 : BOOL ;
   B_Adres_19_bit_3 : BOOL ;
   B_Adres_18_bit_0 : BOOL ;	//Temporary placeholder variable
   B_Adres_18_bit_1 : BOOL ;
   B_Adres_18_bit_2 : BOOL ;
   B_Adres_18_bit_3 : BOOL ;
   B_Adres_21_bit_0 : BOOL ;	//Temporary placeholder variable
   B_Adres_21_bit_1 : BOOL ;
   B_Adres_21_bit_2 : BOOL ;
   B_Adres_21_bit_3 : BOOL ;
   B_Adres_20_bit_0 : BOOL ;	//Temporary placeholder variable
   B_Adres_20_bit_1 : BOOL ;
   B_Adres_20_bit_2 : BOOL ;
   B_Adres_20_bit_3 : BOOL ;
   B_Adres_23_bit_0 : BOOL ;	//Temporary placeholder variable
   B_Adres_23_bit_1 : BOOL ;
   B_Adres_23_bit_2 : BOOL ;
   B_Adres_23_bit_3 : BOOL ;
   B_Adres_22_bit_0 : BOOL ;	//Temporary placeholder variable
   B_Adres_22_bit_1 : BOOL ;
   B_Adres_22_bit_2 : BOOL ;
   B_Adres_22_bit_3 : BOOL ;
   B_Adres_25_bit_0 : BOOL ;	//Temporary placeholder variable
   B_Adres_25_bit_1 : BOOL ;
   B_Adres_25_bit_2 : BOOL ;
   B_Adres_25_bit_3 : BOOL ;
   B_Adres_24_bit_0 : BOOL ;	//Temporary placeholder variable
   B_Adres_24_bit_1 : BOOL ;
   B_Adres_24_bit_2 : BOOL ;
   B_Adres_24_bit_3 : BOOL ;
   B_Adres_27_bit_0 : BOOL ;	//Temporary placeholder variable
   B_Adres_27_bit_1 : BOOL ;
   B_Adres_27_bit_2 : BOOL ;
   B_Adres_27_bit_3 : BOOL ;
   B_Adres_26_bit_0 : BOOL ;	//Temporary placeholder variable
   B_Adres_26_bit_1 : BOOL ;
   B_Adres_26_bit_2 : BOOL ;
   B_Adres_26_bit_3 : BOOL ;
   B_Adres_29_bit_0 : BOOL ;	//Temporary placeholder variable
   B_Adres_29_bit_1 : BOOL ;
   B_Adres_29_bit_2 : BOOL ;
   B_Adres_29_bit_3 : BOOL ;
   B_Adres_28_bit_0 : BOOL ;	//Temporary placeholder variable
   B_Adres_28_bit_1 : BOOL ;
   B_Adres_28_bit_2 : BOOL ;
   B_Adres_28_bit_3 : BOOL ;
   B_Adres_31_bit_0 : BOOL ;	//Temporary placeholder variable
   B_Adres_31_bit_1 : BOOL ;
   B_Adres_31_bit_2 : BOOL ;
   B_Adres_31_bit_3 : BOOL ;
   B_Adres_30_bit_0 : BOOL ;	//Temporary placeholder variable
   B_Adres_30_bit_1 : BOOL ;
   B_Adres_30_bit_2 : BOOL ;
   B_Adres_30_bit_3 : BOOL ;
  END_STRUCT ;	
BEGIN
END_DATA_BLOCK

DATA_BLOCK "Asi_output"	// DB 81
VERSION : 0.1
  STRUCT
   Adres_1_bit_0 : BOOL ;	//Temporary placeholder variable
   Adres_1_bit_1 : BOOL ;
   Adres_1_bit_2 : BOOL ;
   Adres_1_bit_3 : BOOL ;
   Adres_0_bit_0 : BOOL ;	//Temporary placeholder variable
   Adres_0_bit_1 : BOOL ;
   Adres_0_bit_2 : BOOL ;
   Adres_0_bit_3 : BOOL ;
   Adres_3_bit_0 : BOOL ;	//Temporary placeholder variable
   Adres_3_bit_1 : BOOL ;
   Adres_3_bit_2 : BOOL ;
   Adres_3_bit_3 : BOOL ;
   Adres_2_bit_0 : BOOL ;	//Temporary placeholder variable
   Adres_2_bit_1 : BOOL ;
   Adres_2_bit_2 : BOOL ;
   Adres_2_bit_3 : BOOL ;
   Adres_5_bit_0 : BOOL ;	//Temporary placeholder variable
   Adres_5_bit_1 : BOOL ;
   Adres_5_bit_2 : BOOL ;
   Adres_5_bit_3 : BOOL ;
   Adres_4_bit_0 : BOOL ;	//Temporary placeholder variable
   Adres_4_bit_1 : BOOL ;
   Adres_4_bit_2 : BOOL ;
   Adres_4_bit_3 : BOOL ;
   Adres_7_bit_0 : BOOL ;	//Temporary placeholder variable
   Adres_7_bit_1 : BOOL ;
   Adres_7_bit_2 : BOOL ;
   Adres_7_bit_3 : BOOL ;
   Adres_6_bit_0 : BOOL ;	//Temporary placeholder variable
   Adres_6_bit_1 : BOOL ;
   Adres_6_bit_2 : BOOL ;
   Adres_6_bit_3 : BOOL ;
   Adres_9_bit_0 : BOOL ;	//Temporary placeholder variable
   Adres_9_bit_1 : BOOL ;
   Adres_9_bit_2 : BOOL ;
   Adres_9_bit_3 : BOOL ;
   Adres_8_bit_0 : BOOL ;	//Temporary placeholder variable
   Adres_8_bit_1 : BOOL ;
   Adres_8_bit_2 : BOOL ;
   Adres_8_bit_3 : BOOL ;
   Adres_11_bit_0 : BOOL ;	//Temporary placeholder variable
   Adres_11_bit_1 : BOOL ;
   Adres_11_bit_2 : BOOL ;
   Adres_11_bit_3 : BOOL ;
   Adres_10_bit_0 : BOOL ;	//Temporary placeholder variable
   Adres_10_bit_1 : BOOL ;
   Adres_10_bit_2 : BOOL ;
   Adres_10_bit_3 : BOOL ;
   Adres_13_bit_0 : BOOL ;	//Temporary placeholder variable
   Adres_13_bit_1 : BOOL ;
   Adres_13_bit_2 : BOOL ;
   Adres_13_bit_3 : BOOL ;
   Adres_12_bit_0 : BOOL ;	//Temporary placeholder variable
   Adres_12_bit_1 : BOOL ;
   Adres_12_bit_2 : BOOL ;
   Adres_12_bit_3 : BOOL ;
   Adres_15_bit_0 : BOOL ;	//Temporary placeholder variable
   Adres_15_bit_1 : BOOL ;
   Adres_15_bit_2 : BOOL ;
   Adres_15_bit_3 : BOOL ;
   Adres_14_bit_0 : BOOL ;	//Temporary placeholder variable
   Adres_14_bit_1 : BOOL ;
   Adres_14_bit_2 : BOOL ;
   Adres_14_bit_3 : BOOL ;
   Adres_17_bit_0 : BOOL ;	//Temporary placeholder variable
   Adres_17_bit_1 : BOOL ;
   Adres_17_bit_2 : BOOL ;
   Adres_17_bit_3 : BOOL ;
   Adres_16_bit_0 : BOOL ;	//Temporary placeholder variable
   Adres_16_bit_1 : BOOL ;
   Adres_16_bit_2 : BOOL ;
   Adres_16_bit_3 : BOOL ;
   Adres_19_bit_0 : BOOL ;	//Temporary placeholder variable
   Adres_19_bit_1 : BOOL ;
   Adres_19_bit_2 : BOOL ;
   Adres_19_bit_3 : BOOL ;
   Adres_18_bit_0 : BOOL ;	//Temporary placeholder variable
   Adres_18_bit_1 : BOOL ;
   Adres_18_bit_2 : BOOL ;
   Adres_18_bit_3 : BOOL ;
   Adres_21_bit_0 : BOOL ;	//Temporary placeholder variable
   Adres_21_bit_1 : BOOL ;
   Adres_21_bit_2 : BOOL ;
   Adres_21_bit_3 : BOOL ;
   Adres_20_bit_0 : BOOL ;	//Temporary placeholder variable
   Adres_20_bit_1 : BOOL ;
   Adres_20_bit_2 : BOOL ;
   Adres_20_bit_3 : BOOL ;
   Adres_23_bit_0 : BOOL ;	//Temporary placeholder variable
   Adres_23_bit_1 : BOOL ;
   Adres_23_bit_2 : BOOL ;
   Adres_23_bit_3 : BOOL ;
   Adres_22_bit_0 : BOOL ;	//Temporary placeholder variable
   Adres_22_bit_1 : BOOL ;
   Adres_22_bit_2 : BOOL ;
   Adres_22_bit_3 : BOOL ;
   Adres_25_bit_0 : BOOL ;	//Temporary placeholder variable
   Adres_25_bit_1 : BOOL ;
   Adres_25_bit_2 : BOOL ;
   Adres_25_bit_3 : BOOL ;
   Adres_24_bit_0 : BOOL ;	//Temporary placeholder variable
   Adres_24_bit_1 : BOOL ;
   Adres_24_bit_2 : BOOL ;
   Adres_24_bit_3 : BOOL ;
   Adres_27_bit_0 : BOOL ;	//Temporary placeholder variable
   Adres_27_bit_1 : BOOL ;
   Adres_27_bit_2 : BOOL ;
   Adres_27_bit_3 : BOOL ;
   Adres_26_bit_0 : BOOL ;	//Temporary placeholder variable
   Adres_26_bit_1 : BOOL ;
   Adres_26_bit_2 : BOOL ;
   Adres_26_bit_3 : BOOL ;
   Adres_29_bit_0 : BOOL ;	//Temporary placeholder variable
   Adres_29_bit_1 : BOOL ;
   Adres_29_bit_2 : BOOL ;
   Adres_29_bit_3 : BOOL ;
   Adres_28_bit_0 : BOOL ;	//Temporary placeholder variable
   Adres_28_bit_1 : BOOL ;
   Adres_28_bit_2 : BOOL ;
   Adres_28_bit_3 : BOOL ;
   Adres_31_bit_0 : BOOL ;	//Temporary placeholder variable
   Adres_31_bit_1 : BOOL ;
   Adres_31_bit_2 : BOOL ;
   Adres_31_bit_3 : BOOL ;
   Adres_30_bit_0 : BOOL ;	//Temporary placeholder variable
   Adres_30_bit_1 : BOOL ;
   Adres_30_bit_2 : BOOL ;
   Adres_30_bit_3 : BOOL ;
   B_Adres_1_bit_0 : BOOL ;	//Temporary placeholder variable
   B_Adres_1_bit_1 : BOOL ;
   B_Adres_1_bit_2 : BOOL ;
   B_Adres_1_bit_3 : BOOL ;
   B_Adres_0_bit_0 : BOOL ;
   B_Adres_0_bit_1 : BOOL ;
   B_Adres_0_bit_2 : BOOL ;
   B_Adres_0_bit_3 : BOOL ;
   B_Adres_3_bit_0 : BOOL ;	//Temporary placeholder variable
   B_Adres_3_bit_1 : BOOL ;
   B_Adres_3_bit_2 : BOOL ;
   B_Adres_3_bit_3 : BOOL ;
   B_Adres_2_bit_0 : BOOL ;	//Temporary placeholder variable
   B_Adres_2_bit_1 : BOOL ;
   B_Adres_2_bit_2 : BOOL ;
   B_Adres_2_bit_3 : BOOL ;
   B_Adres_5_bit_0 : BOOL ;	//Temporary placeholder variable
   B_Adres_5_bit_1 : BOOL ;
   B_Adres_5_bit_2 : BOOL ;
   B_Adres_5_bit_3 : BOOL ;
   B_Adres_4_bit_0 : BOOL ;	//Temporary placeholder variable
   B_Adres_4_bit_1 : BOOL ;
   B_Adres_4_bit_2 : BOOL ;
   B_Adres_4_bit_3 : BOOL ;
   B_Adres_7_bit_0 : BOOL ;	//Temporary placeholder variable
   B_Adres_7_bit_1 : BOOL ;
   B_Adres_7_bit_2 : BOOL ;
   B_Adres_7_bit_3 : BOOL ;
   B_Adres_6_bit_0 : BOOL ;	//Temporary placeholder variable
   B_Adres_6_bit_1 : BOOL ;
   B_Adres_6_bit_2 : BOOL ;
   B_Adres_6_bit_3 : BOOL ;
   B_Adres_9_bit_0 : BOOL ;	//Temporary placeholder variable
   B_Adres_9_bit_1 : BOOL ;
   B_Adres_9_bit_2 : BOOL ;
   B_Adres_9_bit_3 : BOOL ;
   B_Adres_8_bit_0 : BOOL ;	//Temporary placeholder variable
   B_Adres_8_bit_1 : BOOL ;
   B_Adres_8_bit_2 : BOOL ;
   B_Adres_8_bit_3 : BOOL ;
   B_Adres_11_bit_0 : BOOL ;	//Temporary placeholder variable
   B_Adres_11_bit_1 : BOOL ;
   B_Adres_11_bit_2 : BOOL ;
   B_Adres_11_bit_3 : BOOL ;
   B_Adres_10_bit_0 : BOOL ;	//Temporary placeholder variable
   B_Adres_10_bit_1 : BOOL ;
   B_Adres_10_bit_2 : BOOL ;
   B_Adres_10_bit_3 : BOOL ;
   B_Adres_13_bit_0 : BOOL ;	//Temporary placeholder variable
   B_Adres_13_bit_1 : BOOL ;
   B_Adres_13_bit_2 : BOOL ;
   B_Adres_13_bit_3 : BOOL ;
   B_Adres_12_bit_0 : BOOL ;	//Temporary placeholder variable
   B_Adres_12_bit_1 : BOOL ;
   B_Adres_12_bit_2 : BOOL ;
   B_Adres_12_bit_3 : BOOL ;
   B_Adres_15_bit_0 : BOOL ;	//Temporary placeholder variable
   B_Adres_15_bit_1 : BOOL ;
   B_Adres_15_bit_2 : BOOL ;
   B_Adres_15_bit_3 : BOOL ;
   B_Adres_14_bit_0 : BOOL ;	//Temporary placeholder variable
   B_Adres_14_bit_1 : BOOL ;
   B_Adres_14_bit_2 : BOOL ;
   B_Adres_14_bit_3 : BOOL ;
   B_Adres_17_bit_0 : BOOL ;	//Temporary placeholder variable
   B_Adres_17_bit_1 : BOOL ;
   B_Adres_17_bit_2 : BOOL ;
   B_Adres_17_bit_3 : BOOL ;
   B_Adres_16_bit_0 : BOOL ;	//Temporary placeholder variable
   B_Adres_16_bit_1 : BOOL ;
   B_Adres_16_bit_2 : BOOL ;
   B_Adres_16_bit_3 : BOOL ;
   B_Adres_19_bit_0 : BOOL ;	//Temporary placeholder variable
   B_Adres_19_bit_1 : BOOL ;
   B_Adres_19_bit_2 : BOOL ;
   B_Adres_19_bit_3 : BOOL ;
   B_Adres_18_bit_0 : BOOL ;	//Temporary placeholder variable
   B_Adres_18_bit_1 : BOOL ;
   B_Adres_18_bit_2 : BOOL ;
   B_Adres_18_bit_3 : BOOL ;
   B_Adres_21_bit_0 : BOOL ;	//Temporary placeholder variable
   B_Adres_21_bit_1 : BOOL ;
   B_Adres_21_bit_2 : BOOL ;
   B_Adres_21_bit_3 : BOOL ;
   B_Adres_20_bit_0 : BOOL ;	//Temporary placeholder variable
   B_Adres_20_bit_1 : BOOL ;
   B_Adres_20_bit_2 : BOOL ;
   B_Adres_20_bit_3 : BOOL ;
   B_Adres_23_bit_0 : BOOL ;	//Temporary placeholder variable
   B_Adres_23_bit_1 : BOOL ;
   B_Adres_23_bit_2 : BOOL ;
   B_Adres_23_bit_3 : BOOL ;
   B_Adres_22_bit_0 : BOOL ;	//Temporary placeholder variable
   B_Adres_22_bit_1 : BOOL ;
   B_Adres_22_bit_2 : BOOL ;
   B_Adres_22_bit_3 : BOOL ;
   B_Adres_25_bit_0 : BOOL ;	//Temporary placeholder variable
   B_Adres_25_bit_1 : BOOL ;
   B_Adres_25_bit_2 : BOOL ;
   B_Adres_25_bit_3 : BOOL ;
   B_Adres_24_bit_0 : BOOL ;	//Temporary placeholder variable
   B_Adres_24_bit_1 : BOOL ;
   B_Adres_24_bit_2 : BOOL ;
   B_Adres_24_bit_3 : BOOL ;
   B_Adres_27_bit_0 : BOOL ;	//Temporary placeholder variable
   B_Adres_27_bit_1 : BOOL ;
   B_Adres_27_bit_2 : BOOL ;
   B_Adres_27_bit_3 : BOOL ;
   B_Adres_26_bit_0 : BOOL ;	//Temporary placeholder variable
   B_Adres_26_bit_1 : BOOL ;
   B_Adres_26_bit_2 : BOOL ;
   B_Adres_26_bit_3 : BOOL ;
   B_Adres_29_bit_0 : BOOL ;	//Temporary placeholder variable
   B_Adres_29_bit_1 : BOOL ;
   B_Adres_29_bit_2 : BOOL ;
   B_Adres_29_bit_3 : BOOL ;
   B_Adres_28_bit_0 : BOOL ;	//Temporary placeholder variable
   B_Adres_28_bit_1 : BOOL ;
   B_Adres_28_bit_2 : BOOL ;
   B_Adres_28_bit_3 : BOOL ;
   B_Adres_31_bit_0 : BOOL ;	//Temporary placeholder variable
   B_Adres_31_bit_1 : BOOL ;
   B_Adres_31_bit_2 : BOOL ;
   B_Adres_31_bit_3 : BOOL ;
   B_Adres_30_bit_0 : BOOL ;	//Temporary placeholder variable
   B_Adres_30_bit_1 : BOOL ;
   B_Adres_30_bit_2 : BOOL ;
   B_Adres_30_bit_3 : BOOL ;
  END_STRUCT ;	
BEGIN
END_DATA_BLOCK

DATA_BLOCK "MPI_GD"	// DB 100
VERSION : 0.1
  STRUCT
   IN : STRUCT
    Life_Bit_Foliarka : BOOL ;
    Foliarka_Automatyka : BOOL ;
    Foliarka_Reczny : BOOL ;
    Foto_Banda_1 : BOOL ;
    Foto_Owijarka : BOOL ;
    Rezerwa_1 : BOOL ;
    Motor_10_Lewo : BOOL ;
    Motor_10_Prawo : BOOL ;
    Motor_11_Lewo : BOOL ;
    Motor_11_Prawo : BOOL ;
    Zezwolenie_Na_Wjazd_10 : BOOL ;
    Potw_Dost_Na_Wjazd_10 : BOOL ;
    Zabierz_Na_Bande_11 : BOOL ;
    Paleta_Obecna_Na_7_Tr : BOOL ;
    Help_INT : INT ;
   END_STRUCT ;
   OUT : STRUCT
    Life_Bit_Szafa : BOOL ;
    Szafa_Automatyka : BOOL ;
    Foto_1_Banda_10 : BOOL ;
    Foto_2_Banda_10 : BOOL ;
    Foto_Banda_11 : BOOL ;
    Silnik_10_OK : BOOL ;
    Silnik_11_OK : BOOL ;
    Zabierz_Na_Bande_10 : BOOL ;
    Zezwolenie_Na_Wyjazd_11 : BOOL ;
    Potw_Dost_Na_Wyjazd_11 : BOOL ;
    Obrot_Na_Poz_Wlot_1 : BOOL ;
    Zmien_Program_Na_4 : BOOL ;
    Zmien_Pragram_Na_3 : BOOL ;
    Foto_Banda_9 : BOOL ;
    Help_INT : INT ;
   END_STRUCT ;
  END_STRUCT ;	
BEGIN
END_DATA_BLOCK

DATA_BLOCK "Blok_Bledow"	// DB 119
VERSION : 0.1
  STRUCT
   Blad_Silnika_Adr_1 : BOOL ;	//Blad silnika o adresie 1 - rolki obrotnica bindownicy
   Blad_Silnika_Adr_2 : BOOL ;	//Blad silnika o adresie 2 - rolki wylot bindownicy
   Blad_Silnika_Adr_3 : BOOL ;	//Blad silnika o adresie 3 - rolki
   Blad_Silnika_Adr_4 : BOOL ;	//Blad silnika o adresie 4 - rolki
   Blad_Silnika_Adr_5 : BOOL ;	//Blad silnika o adresie 5 - rolki
   Blad_Silnika_Adr_6 : BOOL ;	//Blad silnika o adresie 6 - rolki
   Blad_Silnika_Adr_7 : BOOL ;	//Blad silnika o adresie 7 - rolki
   Blad_Silnika_Adr_8 : BOOL ;	//Blad silnika o adresie 8 - rolki
   Blad_Silnika_Adr_9 : BOOL ;	//Blad silnika o adresie 9 - rolki
   Blad_Silnika_Adr_10 : BOOL ;	//Blad silnika o adresie 10 - rolki
   Blad_Silnika_Adr_11 : BOOL ;	//Blad silnika o adresie 11 - rolki
   Blad_Silnika_Adr_12 : BOOL ;	//Blad silnika o adresie 12 - rolki
   Blad_Silnika_Adr_13 : BOOL ;	//Blad silnika o adresie 13 - rolki
   Blad_Silnika_Adr_14 : BOOL ;	//Blad silnika o adresie 14 - rolki
   Blad_Silnika_Adr_15 : BOOL ;	//Blad silnika o adresie 15 - silnik obrotnicy bindownicy
   Blad_Rygla_Adr_16 : BOOL ;	//Blad rygla drzwi o adresie 16
   Blad_Silnika_Adr_18 : BOOL ;	//Blad silnika o adresie 18 - silnik obrotnicy wyboru wlotu
   Blad_Silnika_Adr_20 : BOOL ;	//Blad silnika o adresie 20 - silnik obrotnicy etykietownicy
   Blad_Silnika_Adr_23 : BOOL ;	//Blad silnika o adresie 23 - rolki
   Blad_Silnika_Adr_24 : BOOL ;	//Blad silnika o adresie 24 - rolki
   Blad_Kurtyny_Adr_25 : BOOL ;	//Blad kurtyny wlotowej  adres 25
   Blad_Kurtyny_Adr_26 : BOOL ;	//Blad kurtyny wylotowej aders 26
   Blad_Not_Aus_27 : BOOL ;	//Blad Not Aus adres 27 - Not Aus szafa
   Blad_Not_Aus_28 : BOOL ;	//Blad Not Aus adres 28 - Not Aus poczatek lini
   Blad_Not_Aus_29 : BOOL ;	//Blad Not Aus adres 29 - Not Aus srodek lini
   Blad_Not_Aus_30 : BOOL ;	//Blad Not Aus adres 30 - Not Aus koniec lini
   Blad_Not_Aus_31 : BOOL ;	//Blad Not Aus adres 31 - Not Aus panel bindownicy
   Blad_Przek_Bezp_Bind : BOOL ;	//Strefa bezpieczenstwa rejonu bindownicy  niepotwierdzona(wejscie -I4.4)
   Ostrz_Bind_Blad : BOOL ;	//Blad ogolny bindownicy
   Ostrz_Bind_Nie_Cofnieta : BOOL ;	//Bindownica nie jest cofnieta
   Ostrz_Bind_Sygn_Bezp : BOOL ;	//Bindownica brak sygnalu bezpieczenstwa
   Ostrz_Bind_Nie_Jest_Auto : BOOL ;	//Bindownica nie jest w trybie automatycznym (wejscie -I2.4)
   Ostrz_Stol_Obr_Foto : BOOL ;	//Blad fotokomorek stolu obrotowego
   Ostrz_Obr_Stol_Obr_Pozyc : BOOL ;	//Stol obrotowy nie jest w pozycji 0
   Ostrz_Pokr_Foto_Tas_1 : BOOL ;	//Niewlasciwe Pokrycie fotkomorek na tasmie 1 (Przejedz do przodu w recznym )
   Ostrz_Pokr_Foto_Tas_2 : BOOL ;	//Niewlasciwe Pokrycie fotkomorek na tasmie 2 (Przejedz do przodu w recznym )
   Ostrz_Pokr_Foto_Obr : BOOL ;	//Niewlasciwe Pokrycie fotkomorek na obrotnicy (Przejedz do przodu w recznym )
   Ostrz_Pokr_Foto_Tas_4 : BOOL ;	//Niewlasciwe Pokrycie fotkomorek na tasmie 4 (Przejedz do przodu w recznym )
   Blad_Krok_1 : BOOL ;	//Blad kroku nr 1 (Przekrokczony czas jazdy  na zadana pozycje)
   Blad_Krok_2 : BOOL ;	//Blad kroku nr 2 (Przekrokczony czas szukania srodka palety)
   Blad_Krok_3 : BOOL ;	//Blad kroku nr 3 (Przekrokczony czas pozycjonowania palety lewo/prawo)
   Blad_Krok_4 : BOOL ;	//Blad kroku nr 4 (Przekrokczony czas strzalu bindownicy)
   Blad_Krok_5 : BOOL ;	//Blad kroku nr 5 (Przekrokczony czas czasu postoju)
   Blad_Krok_6 : BOOL ;	//Blad kroku nr 6 (Przekrokczony czas powrotu lewo/prawo)
   Alarm_Obr_Stol_Obr_Pozyc : BOOL ;	//Stol obrotowy nie jest w pozycji 0
   Alarm_Bind_Nie_Cofinieta : BOOL ;	//Bindownica nie cofnieta lub brak zezwolenia  (cofnij ramie do tylu)
   Alarm_Bind_Sygn_Bezp : BOOL ;	//Bindownica brak sygnalu bezpieczenstwa
   rez3 : BOOL ;	//rez 3
   rez_6_0 : BOOL ;	//rez_6_0
   Alarm_Pokr_Foto_Tas_1 : BOOL ;	//Niewlasciwe Pokrycie fotkomorek na tasmie 1 (Przejedz do przodu w recznym )
   Alarm_Pokr_Foto_Tas_2 : BOOL ;	//Niewlasciwe Pokrycie fotkomorek na tasmie 2 (Przejedz do przodu w recznym )
   Alarm_Pokr_Foto_Tas_4 : BOOL ;	//Niewlasciwe Pokrycie fotkomorek na tasmie 4 (Przejedz do przodu w recznym )
   Alarm_Pokr_Foto_Obr : BOOL ;	//Niewlasciwe Pokrycie fotkomorek na obrotnicy przy braku cyklu
   Alarm_Bind_Nie_Jest_Auto : BOOL ;	//Bindownica nie jest w trybie automatycznym (wejscie -I2.4)
   Alarm_Bind_Blad : BOOL ;	//Blad ogolny bindownicy
   rez_6_7 : BOOL ;	//rez_6_7
   Ostrz_Prasa_Nie_W_Gorze : BOOL ;	//Zlamywak dekli nie jest u gory I2.6
   rez_7_1 : BOOL ;	//rez_7_1
   rez_7_2 : BOOL ;	//rez_7_2
   rez_7_3 : BOOL ;	//rez_7_3
   rez_7_4 : BOOL ;	//rez_7_4
   rez_7_5 : BOOL ;	//rez_7_5
   Ostrz_Wozek_Przy_Przen : BOOL ;	//Wozek widlowy przy przenosniku (i2.7)
   Ostrz_C_Bind_Foto_Pokr : BOOL ;	//Pokrycie fotokomorek podczas cyklu bindowania
   Ostrz_C_Bind_Poz_Bindow : BOOL ;	//Pozycja bindownicy podczas bindowania
   rez_8_1 : BOOL ;	//rez_8_1
   rez_8_2 : BOOL ;	//rez_8_2
   rez_8_3 : BOOL ;	//rez_8_3
   rez_8_4 : BOOL ;	//rez_8_4
   rez_8_5 : BOOL ;	//rez_8_5
   rez_8_6 : BOOL ;	//rez_8_6
   rez_8_7 : BOOL ;	//rez_8_7
   rez_9_0 : BOOL ;	//rez_9_0
   rez_9_1 : BOOL ;	//rez_9_1
   rez_9_2 : BOOL ;	//rez_9_2
   rez_9_3 : BOOL ;	//rez_9_3
   rez_9_4 : BOOL ;	//rez_9_4
   rez_9_5 : BOOL ;	//rez_9_5
   rez_9_6 : BOOL ;	//rez_9_6
   rez_9_7 : BOOL ;	//rez_9_7
   rez_int_bl : INT ;
   rez_int_bl_2 : INT ;
  END_STRUCT ;	
BEGIN
END_DATA_BLOCK

DATA_BLOCK "DB_HMI"	// DB 120
VERSION : 0.1
  STRUCT
   HMI_IN : STRUCT 	//Zmienne wchodzace do HMI nie nadpisywane W HMI (100 bajtow)
    Tryb_Reczny : BOOL ;	//Tryb Reczny
    Tryb_Auto : BOOL ;	//Tryb Auto
    Pozycja_0_st : BOOL ;	//Obrotnica Pozycja 0 st
    Pozycja_90_st : BOOL ;	//Obrotnica Pozycja 90 st
    Pozycja_180_st : BOOL ;	//Obrotnica Pozycja 180 st
    Pozycja_270_st : BOOL ;	//Obrotnica Pozycja 270 st
    Foto_Tasma_1_Tyl : BOOL ;	//foto tylne na bandzie wlotowej
    Foto_Tasma_1_Przod : BOOL ;	//foto przednie bandzie wlotowej
    Foto_Tasma_2_Tyl : BOOL ;	//foto tylne na bandzie wlotowej 2
    Foto_Tasma_2_Przod : BOOL ;	//foto przednie na bandzie wlotowej 2
    Foto_Obrotnica_3_Tyl : BOOL ;	//foto tylne na obrotnicy 3
    Foto_Obrotnica_3_Przod : BOOL ;	//foto przednie na obrotnicy 3
    Foto_Tasma_4_Tyl : BOOL ;	//foto tylne na bandzie wylotowej 4
    Foto_Tasma_4_Przod : BOOL ;	//foto przednie na bandzie wlotowej 4
    Motor_Tasma_1_Tyl : BOOL ;	//motor tasma 1 tyl
    Motor_Tasma_1_Przod : BOOL ;	//motor tasma 1 przod
    Motor_Tasma_2_Tyl : BOOL ;	//motor tasma 2 tyl
    Motor_Tasma_2_Przod : BOOL ;	//motor tasma 2 przod
    Motor_Tasma_3_Tyl : BOOL ;	//motor tasma obrotnica 3 tyl
    Motor_Tasma_3_Przod : BOOL ;	//motor tasma obrotnica 3 przod
    Motor_Obrotnica_3_CW : BOOL ;	//motor obrotnica 3 clock wise
    Motor_Obrotnica_3_CCW : BOOL ;	//motor obrotnica 3 counter clock wise
    Motor_Tasma_4_Przod : BOOL ;	//motor tasma obrotnica 4 tyl
    Motor_Tasma_4_Tyl : BOOL ;	//motor tasma obrotnica 4 przod
    Kurtyna_Wlot_Ok : BOOL ;	//kurtyna na wlocie ok
    Kurtyna_Wylot_Ok : BOOL ;	//kurtyna na wylocie ok
    Wybrano_TP_Przelot : BOOL ;	//wybrano tryb pracy przelot
    Wybrano_TP_Wiazanie_Wzdl : BOOL ;	//wybrano tryb pracy wiazanie wzdluzne
    Wybrano_TP_Wiazanie_Pop : BOOL ;	//wybrano tryb pracy wiazanie poprzeczne
    Wybrano_TP_Wiazanie_Krzy : BOOL ;	//wybrano tryb pracy wiazanie krzyzowe
    Czujnik_Ham_0_St : BOOL ;	//fotokomorka hamowania obrotnicy do kata 0st
    Czujnik_0_St : BOOL ;	//fotokomorka zatrzymania obrotnicy przy kacie 0st
    Czujnik_Ham_90_St : BOOL ;	//fotokomorka hamowania obrotnicy do kata 90st
    Czujnik_90_St : BOOL ;	//fotokomorka zatrzymania obrotnicy przy kacie 90st
    Czujnik_Ham_180_St : BOOL ;	//fotokomorka hamowania obrotnicy do kata 180st
    Czujnik_180_St : BOOL ;	//fotokomorka zatrzymania obrotnicy przy kacie 180st
    Czujnik_Ham_270_St : BOOL ;	//fotokomorka hamowania obrotnicy do kata 270st
    Czujnik_270_St : BOOL ;	//fotokomorka zatrzymania obrotnicy przy kacie 270st
    Interfefs_B_do_TP_B1 : BOOL ;	//obwod bezpieczenstwa bindownicy
    Interfefs_B_do_TP_B2 : BOOL ;	//polozenie podstawowe bindownicy
    Interfefs_B_do_TP_B3 : BOOL ;	//start/zakonczenie wiazania
    Interfefs_B_do_TP_B5 : BOOL ;	//blad bindownicy
    Interfefs_TP_do_B_TP1 : BOOL ;	//obwod bezpieczenstwa tasmociagow
    Interfefs_TP_do_B_TP2 : BOOL ;	//zezwolenie na prace bindownicy
    Interfefs_TP_do_B_TP3 : BOOL ;	//start wiazania
    PB_Strefa_bezpieczenstwa : BOOL ;	//przycisk zalaczenie Strefy bezpieczenstwa
    PB_Reczny : BOOL ;	//przycisk trybu reczny
    PB_Auto : BOOL ;	//przycisk auto
    PB_Reset : BOOL ;	//przycisk reset
    PB_Stop : BOOL ;	//przycisk stop
    PB_Cykl_Start : BOOL ;	//przycisk start cyklu
    PB_Tasma1_Tyl : BOOL ;	//przycisk tasma 1 do tylu
    PB_Tasma1_Przod : BOOL ;	//przycisk tasma 1 do przodu
    PB_Tasma2_Tyl : BOOL ;	//przycisk tasma 2 do tylu
    PB_Tasma2_Przod : BOOL ;	//przycisk tasma 2 do przodu
    PB_Tasma3_Tyl : BOOL ;	//przycisk tasma 3 do tylu
    PB_Tasma3_Przod : BOOL ;	//przycisk tasma 3 do przodu
    PB_Tasma4_Tyl : BOOL ;	//przycisk tasma 4 do tylu
    PB_Tasma4_Przod : BOOL ;	//przycisk tasma 4 do przodu
    PB_Tasma3_Obr_CW : BOOL ;	//przycisk obrotnica w prawo
    PB_Tasma3_Obr_CCW : BOOL ;	//przycisk obrotnica w lewo
    Lampka_Blad_Bind : BOOL ;	//lamka bledu bindownicy
    Lampka_Strzal_Tasmy : BOOL ;	//lampka wystrzalu tasmy
    Lampka_Strefa_Bezp : BOOL ;	//lampka przycisku strefy bezpieczenstwa
    Lampka_PB_Reczny : BOOL ;	//lampka przycisku trybu recznego
    Lampka_PB_Auto : BOOL ;	//lampka przycisku trybu auto
    Lampka_PB_Reset : BOOL ;	//lampka przycisku reset
    Lampka_PB_Stop : BOOL ;	//lampka przycisku stop
    Lampka_PB_Cykl_Start : BOOL ;	//lampka przycisku start
    Paleta_na_Tasmie_1 : BOOL ;	//znacznik palety na tasmie 1
    Paleta_na_Tasmie_2 : BOOL ;	//znacznik palety na tasmie 2
    Paleta_na_Tasmie_3_0_180 : BOOL ;	//znacznik palety na tasmie 3 przy kacie 0 lub 180st
    Paleta_na_Tasmie_3_90_27 : BOOL ;	//znacznik palety na tasmie 3 przy kacie 90 lub 270st
    Paleta_na_Tasmie_4 : BOOL ;	//znacznik palety na tasmie 4
    Paleta_na_Tasmie_1_T : BOOL ;	//znacznik palety na tasmie 1 wjazd
    Paleta_na_Tasmie_1_P : BOOL ;	//znacznik palety na tasmie 1 wyjazd
    Paleta_na_Tasmie_2_T : BOOL ;	//znacznik palety na tasmie 2 wjazd
    Paleta_na_Tasmie_2_P : BOOL ;	//znacznik palety na tasmie 2 wyjazd
    Paleta_na_Tasmie_3_T : BOOL ;	//znacznik palety na tasmie 3 wjazd
    Paleta_na_Tasmie_3_P : BOOL ;	//znacznik palety na tasmie 3 wyjazd
    Paleta_na_Tasmie_4_T : BOOL ;	//znacznik palety na tasmie 4 wjazd
    Paleta_na_Tasmie_4_P : BOOL ;	//znacznik palety na tasmie 4 wyjazd
    Rygiel : BOOL ;	//znacznik rygla drzwi
    Blad : BOOL ;	//Znacznik bledu
    Linia_transportowa_praca : BOOL ;	//Znacznik pracy calej linii transportowej
    Interfefs_B_do_TP_B4 : BOOL ;	//tryb pracy bindownicy: Auto(1) Reczny(0)
    Krok_1 : BOOL ;	//krok 1 trybu pracy
    Krok_2 : BOOL ;	//krok 2 trybu pracy
    Krok_3 : BOOL ;	//krok 3 trybu pracy
    Krok_4 : BOOL ;	//krok 4 trybu pracy
    Krok_5 : BOOL ;	//krok 5 trybu pracy
    Krok_6 : BOOL ;	//krok 6 trybu pracy
    Znacznik_Migania_Bledu : BOOL ;	//znacznik migania bledu
    Czujnik_Prasa : BOOL ;	//czujnik prasy s 22
    Stan_Zaworu : BOOL ;
    Tablica_IN_bool : ARRAY  [1 .. 10 ] OF BOOL  := FALSE;
    Tablica_IN_Byte : ARRAY  [1 .. 6 ] OF BYTE  := B#16#0;
    input_0 : BYTE ;
    input_1 : BYTE ;
    input_2 : BYTE ;
    input_3 : BYTE ;
    output_0 : BYTE ;
    output_1 : BYTE ;
    output_2 : BYTE ;
    output_3 : BYTE ;
    input_8 : BYTE ;
    input_9 : BYTE ;
    input_10 : BYTE ;
    input_11 : BYTE ;
    Tablica_IN_DWORD : ARRAY  [1 .. 4 ] OF DWORD ;
    NR_Kroku : DINT ;	//Numer kroku
    Aktualna_Data : DATE_AND_TIME ;
    Tablica_IN_INT : ARRAY  [1 .. 18 ] OF INT ;
    tryb_wiaz : INT ;	//znacznik wyboru trybu wiazania
    INT_Liczba_Akt_Kroku : INT ;	//znacznik wyboru aktualnie wykonywanego kroku
   END_STRUCT ;
   HMI_OUT : STRUCT 	//Zmienne wychodzace z HMI Nie nadpisywane w sterowniku od 100 bajta
    Rezerwa_Out_1 : BOOL ;
    Rezerwa_Out_2 : BOOL ;
    Start_Lini_z_OP : BOOL ;	//start calej lini z HMI
    Stop_Lini_z_OP : BOOL ;	//stop calej lini z HMI
    Wyzwolenie_Wyjazdu : BOOL ;	//wyzwolenie wyjazdu palety na stanowisku bindujacym (tylko w auto)
    Przycisk_Test_Lampek : BOOL ;	//przycisk test lampek
    Przycisk_Reset_Bledow : BOOL ;	//Przycisk resetowania bledow na panelu HMI
    Przycisk_Pozycjonowanie : BOOL ;	//Przycisk HMI do pozycjonowania palety
    H_Zalacz_Zawor_Prasa : BOOL ;	//Zalacz zawor prasa
    H_Zezwl_Ekran_Prasa : BOOL ;	//Zezwolenie na prase reczny
    Tablica_OUT_Bool : ARRAY  [1 .. 144 ] OF BOOL ;
    Tablina_OUT_INT : ARRAY  [1 .. 40 ] OF INT ;
   END_STRUCT ;
   HMI_IN_OUT : STRUCT 	//Zmienne nadpisywane w sterowniku i w HMI od 200 bajta
    Rezerwa_IN_Out_1 : BOOL ;
    Tp_Przelot : BOOL ;	//Tryb Pracy Przelot
    Tp_Wiazanie_Poprzeczne : BOOL ;	//Tryb Pracy Wiazanie poprzeczne
    Tp_Wiazanie_Wzdluzne : BOOL ;	//Tryb Pracy Wiazanie wzduzne
    Tp_Wiazanie_Pop_Wzdl : BOOL ;	//Tryb Pracy Wiaznie Poprzeczne i wzdluzne
    Tp_Pozycjonowanie : BOOL ;	//Tryb Pracy Pozycjonowanie Palety zalaczone
    Test_Lampek : BOOL ;	//Test Lampek
    Reset_bledow : BOOL ;	//Reset Bledow
    Zlamywak_Dekl : BOOL ;	//lamanie dekli
    Tablica_IN_OUT_Bool : ARRAY  [1 .. 144 ] OF BOOL ;
    Tablica_IN_OUT_INT : ARRAY  [1 .. 40 ] OF INT ;
    Wybor_trybu_pracy : BYTE ;
   END_STRUCT ;
  END_STRUCT ;	
BEGIN
   HMI_IN.Foto_Obrotnica_3_Przod := TRUE;
END_DATA_BLOCK

ORGANIZATION_BLOCK OB 1
TITLE = "Main Program Sweep (Cycle)"
VERSION : 0.1
VAR_TEMP
  OB1_EV_CLASS : BYTE ;	//Bits 0-3 = 1 (Coming event), Bits 4-7 = 1 (Event class 1)
  OB1_SCAN_1 : BYTE ;	//1 (Cold restart scan 1 of OB 1), 3 (Scan 2-n of OB 1)
  OB1_PRIORITY : BYTE ;	//Priority of OB Execution
  OB1_OB_NUMBR : BYTE ;	//1 (Organization block 1, OB1)
  OB1_RESERVED_1 : BYTE ;	//Reserved for system
  OB1_RESERVED_2 : BYTE ;	//Reserved for system
  OB1_PREV_CYCLE : INT ;	//Cycle time of previous OB1 scan (milliseconds)
  OB1_MIN_CYCLE : INT ;	//Minimum cycle time of OB1 (milliseconds)
  OB1_MAX_CYCLE : INT ;	//Maximum cycle time of OB1 (milliseconds)
  OB1_DATE_TIME : DATE_AND_TIME ;	//Date and time OB1 started
END_VAR
BEGIN
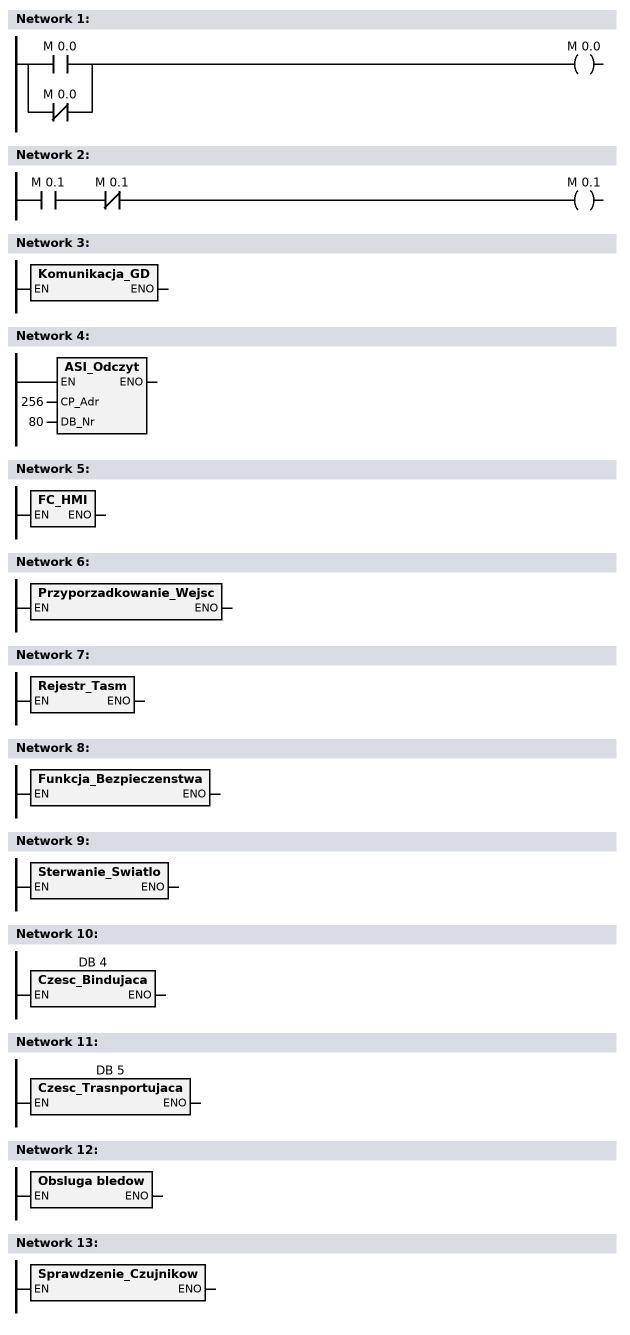
NETWORK
TITLE =
//Zawsze true
      O     M 0.0;
      ON    M 0.0;
      =     M 0.0;
NETWORK
TITLE =
//Zawsze False
      A     M 0.1;
      AN    M 0.1;
      =     M 0.1;
NETWORK
TITLE =
//   BEU   
      CALL  "Komunikacja_GD";
      NOP   0;
NETWORK
TITLE =
//Odczyt wejsc ASI
      CALL  "ASI_Odczyt" (
           CP_Adr                   := 256,
           DB_Nr                    := 80);
      NOP   0;
NETWORK
TITLE =
//komunikacja z hmi
      CALL  "FC_HMI";
      NOP   0;
NETWORK
TITLE =
      CALL  "Przyporzadkowanie_Wejsc";
      NOP   0;
NETWORK
TITLE =
      CALL  "Rejestr_Tasm";
      NOP   0;
NETWORK
TITLE =
      CALL  "Funkcja_Bezpieczenstwa";
      NOP   0;
NETWORK
TITLE =
      CALL  "Sterwanie_Swiatlo";
      NOP   0;
NETWORK
TITLE =
      CALL  "Czesc_Bindujaca" , DB 4;
      NOP   0;
NETWORK
TITLE =
      CALL  "Czesc_Trasnportujaca" , DB 5;
      NOP   0;
NETWORK
TITLE =
      CALL  "Obsluga bledow";
      NOP   0;
NETWORK
TITLE =
      CALL  "Sprawdzenie_Czujnikow";
      NOP   0;
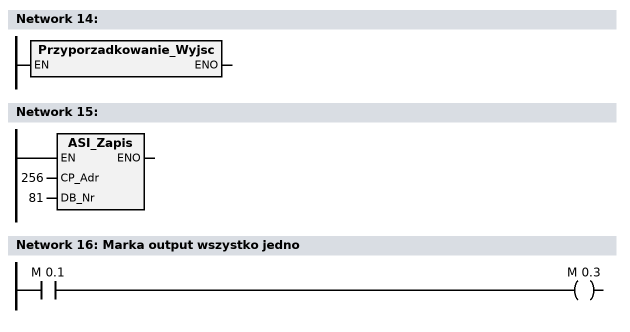
NETWORK
TITLE =
      CALL  "Przyporzadkowanie_Wyjsc";
      NOP   0;
NETWORK
TITLE =
      CALL  "ASI_Zapis" (
           CP_Adr                   := 256,
           DB_Nr                    := 81);
      NOP   0;
NETWORK
TITLE = Marka output wszystko jedno
      A     M 0.1;
      =     M 0.3;
NETWORK
TITLE =
END_ORGANIZATION_BLOCK

ORGANIZATION_BLOCK "I/O_FLT1"	// OB 82
TITLE = "I/O Point Fault"
VERSION : 0.1
VAR_TEMP
  OB82_EV_CLASS : BYTE ;	//16#39, Event class 3, Entering event state, Internal fault event
  OB82_FLT_ID : BYTE ;	//16#XX, Fault identifcation code
  OB82_PRIORITY : BYTE ;	//Priority of OB Execution
  OB82_OB_NUMBR : BYTE ;	//82 (Organization block 82, OB82)
  OB82_RESERVED_1 : BYTE ;	//Reserved for system
  OB82_IO_FLAG : BYTE ;	//Input (01010100), Output (01010101)
  OB82_MDL_ADDR : WORD ;	//Base address of module with fault
  OB82_MDL_DEFECT : BOOL ;	//Module defective
  OB82_INT_FAULT : BOOL ;	//Internal fault
  OB82_EXT_FAULT : BOOL ;	//External fault
  OB82_PNT_INFO : BOOL ;	//Point information
  OB82_EXT_VOLTAGE : BOOL ;	//External voltage low
  OB82_FLD_CONNCTR : BOOL ;	//Field wiring connector missing
  OB82_NO_CONFIG : BOOL ;	//Module has no configuration data
  OB82_CONFIG_ERR : BOOL ;	//Module has configuration error
  OB82_MDL_TYPE : BYTE ;	//Type of module
  OB82_SUB_MDL_ERR : BOOL ;	//Sub-Module is missing or has error
  OB82_COMM_FAULT : BOOL ;	//Communication fault
  OB82_MDL_STOP : BOOL ;	//Module is stopped
  OB82_WTCH_DOG_FLT : BOOL ;	//Watch dog timer stopped module
  OB82_INT_PS_FLT : BOOL ;	//Internal power supply fault
  OB82_PRIM_BATT_FLT : BOOL ;	//Primary battery is in fault
  OB82_BCKUP_BATT_FLT : BOOL ;	//Backup battery is in fault
  OB82_RESERVED_2 : BOOL ;	//Reserved for system
  OB82_RACK_FLT : BOOL ;	//Rack fault, only for bus interface module
  OB82_PROC_FLT : BOOL ;	//Processor fault
  OB82_EPROM_FLT : BOOL ;	//EPROM fault
  OB82_RAM_FLT : BOOL ;	//RAM fault
  OB82_ADU_FLT : BOOL ;	//ADU fault
  OB82_FUSE_FLT : BOOL ;	//Fuse fault
  OB82_HW_INTR_FLT : BOOL ;	//Hardware interupt input in fault
  OB82_RESERVED_3 : BOOL ;	//Reserved for system
  OB82_DATE_TIME : DATE_AND_TIME ;	//Date and time OB82 started
END_VAR
BEGIN
NETWORK
TITLE =
END_ORGANIZATION_BLOCK

ORGANIZATION_BLOCK "RACK_FLT"	// OB 86
TITLE = "Loss Of Rack Fault"
VERSION : 0.1
VAR_TEMP
  OB86_EV_CLASS : BYTE ;	//16#38/39 Event class 3
  OB86_FLT_ID : BYTE ;	//16#C1/C4/C5, Fault identifcation code
  OB86_PRIORITY : BYTE ;	//Priority of OB Execution
  OB86_OB_NUMBR : BYTE ;	//86 (Organization block 86, OB86)
  OB86_RESERVED_1 : BYTE ;	//Reserved for system
  OB86_RESERVED_2 : BYTE ;	//Reserved for system
  OB86_MDL_ADDR : WORD ;	//Base address of IM module in rack with fault
  OB86_RACKS_FLTD : ARRAY  [0 .. 31 ] OF BOOL ;	//Racks in fault
  OB86_DATE_TIME : DATE_AND_TIME ;	//Date and time OB86 started
END_VAR
BEGIN
// (block stored without names or comments; labels and parameter names are numbered)
END_ORGANIZATION_BLOCK

ORGANIZATION_BLOCK "COMPLETE RESTART"	// OB 100
TITLE = "Complete Restart"
VERSION : 0.1
VAR_TEMP
  OB100_EV_CLASS : BYTE ;	//16#13, Event class 1, Entering event state, Event logged in diagnostic buffer
  OB100_STRTUP : BYTE ;	//16#81/82/83/84 Method of startup
  OB100_PRIORITY : BYTE ;	//Priority of OB Execution
  OB100_OB_NUMBR : BYTE ;	//100 (Organization block 100, OB100)
  OB100_RESERVED_1 : BYTE ;	//Reserved for system
  OB100_RESERVED_2 : BYTE ;	//Reserved for system
  OB100_STOP : WORD ;	//Event that caused CPU to stop (16#4xxx)
  OB100_STRT_INFO : DWORD ;	//Information on how system started
  OB100_DATE_TIME : DATE_AND_TIME ;	//Date and time OB100 started
END_VAR
BEGIN
NETWORK
TITLE =
END_ORGANIZATION_BLOCK

ORGANIZATION_BLOCK "PROG_ERR"	// OB 121
TITLE = "Programming Error"
VERSION : 0.1
VAR_TEMP
  OB121_EV_CLASS : BYTE ;	//16#25, Event class 2, Entering event state, Internal fault event
  OB121_SW_FLT : BYTE ;	//16#XX Software programming fault
  OB121_PRIORITY : BYTE ;	//Priority of OB Execution
  OB121_OB_NUMBR : BYTE ;	//121 (Organization block 121, OB121)
  OB121_BLK_TYPE : BYTE ;	//16#88/8A/8B/8C/8E Type of block fault occured in
  OB121_RESERVED_1 : BYTE ;	//Reserved for system
  OB121_FLT_REG : WORD ;	//16#XX Specific register that caused fault
  OB121_BLK_NUM : WORD ;	//Number of block that programming fault occured in
  OB121_PRG_ADDR : WORD ;	//Address in block where programming fault occured
  OB121_DATE_TIME : DATE_AND_TIME ;	//Date and time OB121 started
END_VAR
BEGIN
NETWORK
TITLE =
END_ORGANIZATION_BLOCK
